{attribute 'qualified_only'}
VAR_GLOBAL
END_VAR

(* stored: Version 1.1.0.1, ProductVersion 3.1.4022.7
   GVL GVL_02_Parameter_Step_Motor_BOX_X: Id {bc6c15ad-a728-4b16-bd69-b79c0b13714c} *)
